{attribute 'linkalways'} 
{attribute 'no_explicit_call' := 'This FB is a CLASS and must be accessed using methods or properties'}
{attribute 'enable_dynamic_creation'}
FUNCTION_BLOCK _ETcVnPixelConnectivity EXTENDS EnumDatatypeBase
VAR
	localData : ETcVnPixelConnectivity;
	activeData : REFERENCE TO ETcVnPixelConnectivity;
	enumBaseDatatype : _DINT(localData);
END_VAR

METHOD PRIVATE AddLocalEnumeration
VAR_INPUT
	Enumeration : T_MAXSTRING;
	Value : ETcVnPixelConnectivity;
END_VAR
AddEnumeration(Enumeration, Value);
END_METHOD

PROPERTY PUBLIC Address : PVOID
GET
Address := ADR(activeData);
END_GET
END_PROPERTY

METHOD PUBLIC ClearReference
VAR_INPUT
END_VAR
activeData REF= localData;
SetBaseDatatypeReference();
END_METHOD

METHOD PUBLIC Clone : I_Datatype
VAR
    pClone : POINTER TO _ETcVnPixelConnectivity;
END_VAR
pClone := __NEW(_ETcVnPixelConnectivity(InitialValue := Value));
Clone := pClone^;
END_METHOD

METHOD FB_init : BOOL
VAR_INPUT
	bInitRetains : BOOL; // if TRUE, the retain variables are initialized (warm start / cold start)
	bInCopyCode : BOOL;  // if TRUE, the instance afterwards gets moved into the copy code (online change)
	InitialValue : ETcVnPixelConnectivity;
END_VAR
localData := InitialValue;
AddBaseDatatype(enumBaseDatatype);
ClearReference();

AddLocalEnumeration('TCVN_PC_4', ETcVnPixelConnectivity.TCVN_PC_4);
AddLocalEnumeration('TCVN_PC_8', ETcVnPixelConnectivity.TCVN_PC_8);
END_METHOD

PROPERTY PUBLIC Identifier : T_MAXSTRING
GET
Identifier := 'ETcVnPixelConnectivity';
END_GET
END_PROPERTY

METHOD IsEnumeratorValueEqual : BOOL
VAR_INPUT
	Enumerator : I_KeyValueForwardEnumerator;
END_VAR
VAR
	storedValue : ETcVnPixelConnectivity;
END_VAR
IF NOT Enumerator.TryGet(storedValue) THEN
	RETURN;
END_IF

IsEnumeratorValueEqual := storedValue = activeData;
END_METHOD

METHOD PUBLIC MakeReferenceTo
VAR_INPUT
	ReferenceTarget : REFERENCE TO ETcVnPixelConnectivity;
END_VAR
activeData REF= ReferenceTarget;
SetBaseDatatypeReference();
END_METHOD

METHOD PROTECTED SetBaseDatatypeReference
VAR_INPUT
END_VAR
enumBaseDatatype.MakeReferenceTo(activeData);
END_METHOD

PROPERTY PUBLIC Size : UDINT
GET
Size := SIZEOF(activeData);
END_GET
END_PROPERTY

METHOD TryMakeReferenceTo : BOOL
VAR_INPUT
	Target : I_Datatype;
END_VAR
VAR
	targetAsEnum : I_EnumDatatype;
	pTargetData : POINTER TO ETcVnPixelConnectivity;
END_VAR
IF NOT Target.TryResolveAsEnumDatatype(targetAsEnum) THEN
	RETURN;
END_IF

IF targetAsEnum.Identifier <> Identifier THEN
	RETURN;
END_IF

pTargetData := Target.Address;
activeData REF= pTargetData^;
SetBaseDatatypeReference();
TryMakeReferenceTo := TRUE;
END_METHOD

PROPERTY PUBLIC Value : ETcVnPixelConnectivity
GET
Value := activeData;
END_GET
SET
activeData := Value;
END_SET
END_PROPERTY

END_FUNCTION_BLOCK

(* stored: Version 1.1.0.1, ProductVersion 3.1.4024.12
   POU _ETcVnPixelConnectivity: Id {9adcdad0-0816-46e3-a0b7-a90030c29e79}, SpecialFunc None
   Folder Constructor: Id {ba840882-7e8c-4911-a41d-fa1d24af4319}
   Folder Private: Id {ee73937d-fe72-4a30-ab37-0430ff1c7d32}
   Folder Protected: Id {14e5370b-cd28-4056-949e-7de5e74f7672}
   Method AddLocalEnumeration: Id {fb11d33f-3693-49b0-8bc7-261f5728b902}
   Property Address: Id {0e577a86-5e56-4e23-8834-a7a97e19ba92}
   Get Get: Id {75da68fe-746f-4fb6-9c71-0f6e978b1ef5}
   Method ClearReference: Id {36f3d685-77b7-4051-809a-a4e82c3a7e4c}
   Method Clone: Id {b6dee889-9318-4eb5-b71a-75b58162028a}
   Method FB_init: Id {eb8f3be5-4555-4532-9dbc-485e17d3a14c}
   Property Identifier: Id {ae712f1e-89a9-4e15-aeab-48e1e012194b}
   Get Get: Id {0b495149-cb75-4532-8154-ade9d815d7fc}
   Method IsEnumeratorValueEqual: Id {1dc11014-63a0-4a94-b9f9-e057ef62863c}
   Method MakeReferenceTo: Id {be69636c-61bc-4968-882b-9ce609217f60}
   Method SetBaseDatatypeReference: Id {52597639-8574-4813-96ab-76ae557704db}
   Property Size: Id {6a928913-d683-4baa-8885-38f085dbda8d}
   Get Get: Id {22ee9990-7677-457d-896b-b418b1a24bec}
   Method TryMakeReferenceTo: Id {f30dc729-d5b8-48d5-bf29-bf5db4d4373c}
   Property Value: Id {ebfb50b3-9f82-4760-84bb-6fbe55fc3df4}
   Get Get: Id {4f647025-7b2b-4182-894c-69c89b5d89f0}
   Set Set: Id {92eaeeef-93e2-41f0-9aed-4694d7fc1540} *)
